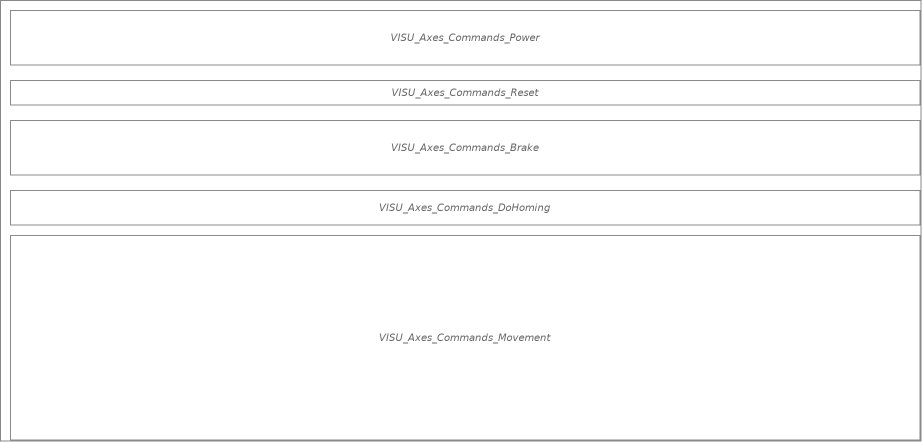
VISUALIZATION VISU_AxesAzimuthAxis_Processes  // 922x442
VAR_IN_OUT
	ref : AxesAzimuthAxis;
    ref_aziDriveChannel : AX52XXDriveChannel;
    widget : AxesAzimuthAxisWidget;
END_VAR
    Frame (10,10 910x55)
        shows VISU_Axes_Commands_Power(powerOn := ref.processes.powerOn, powerOff := ref.processes.powerOff, powerOnStatus := widget.processes_powerOnStatus, powerOffStatus := widget.processes_powerOffStatus)
    Frame (10,80 910x25)
        shows VISU_Axes_Commands_Reset(reset := ref.processes.reset, resetStatus := widget.processes_resetStatus)
    Frame (10,120 910x55)
        shows VISU_Axes_Commands_Brake(unlockBrake := ref.processes.unlockBrake, setBrake := ref_aziDriveChannel.processes.setBrake, unlockBrakeStatus := widget.processes_unlockBrakeStatus, setBrakeStatus := widget.aziDriveChannel.processes_setBrakeStatus)
    Frame (10,190 910x35)
        shows VISU_Axes_Commands_DoHoming(doHoming := ref.processes.doHoming, doHomingStatus := widget.processes_doHomingStatus)
    Frame (10,235 910x205)
        shows VISU_Axes_Commands_Movement(stop := ref.processes.stop, moveOutOfLimitSwitch := ref.processes.moveOutOfLimitSwitch, moveAbsolute := ref.processes.moveAbsolute, moveRelative := ref.processes.moveRelative, moveVelocity := ref.processes.moveVelocity, stopStatus := widget.processes_stopStatus, moveOutOfLimitSwitchStatus := widget.processes_moveOutOfLimitSwitchStatus, moveAbsoluteStatus := widget.processes_moveAbsoluteStatus, moveRelativeStatus := widget.processes_moveRelativeStatus, moveVelocityStatus := widget.processes_moveVelocityStatus)
END_VISUALIZATION

(* stored: Version 1.1.0.1, ProductVersion 3.1.4019.2
   Visu VISU_AxesAzimuthAxis_Processes: Id {2d5b0c93-aad6-4085-9ebd-f7ca15219210} *)
